// TIA Portal V17 export
// export: Created 2026-04-13T11:12:53.7703103Z, ExportSetting WithDefaults, DisplayName Totally Integrated Automation Portal, DisplayVersion V17 Update 4, DisplayName TIA Portal Openness, DisplayVersion V17 Update 4, DisplayName TIA Portal Version Control Interface, DisplayVersion V17, DisplayName SINAMICS Startdrive Advanced, DisplayVersion V17, DisplayName SINAMICS Startdrive G130, G150, S120, S150, SINAMICS MV, S210, DisplayVersion V17, DisplayName SINAMICS Startdrive G110M, G120, G120C, G120D, G120P, G115D, DisplayVersion V17, DisplayName STEP 7 Professional, DisplayVersion V17 Update 4, DisplayName STEP 7 Safety, DisplayVersion V17, DisplayName WinCC Professional, DisplayVersion V17 Update 4
TagTable "PV"
  PV_JF进风温度 : Real  (PLC tag PV.JF进风温度, HMI_连接_1, 1 s)
  PV_JF进风温度写读 : Real  (PLC tag PV.JF进风温度写读, HMI_连接_1, 1 s)
  PV_CF出风温度 : Real  (PLC tag PV.CF出风温度, HMI_连接_1, 1 s)
  PV_WQ尾气温度 : Real  (PLC tag PV.WQ尾气温度, HMI_连接_1, 1 s)
  PV_JF进风温度P : Real  (PLC tag PV.JF进风温度P, HMI_连接_1, 1 s)
  PV_JF进风温度I : Real  (PLC tag PV.JF进风温度I, HMI_连接_1, 1 s)
  PV_JF进风温度D : Real  (PLC tag PV.JF进风温度D, HMI_连接_1, 1 s)
  PV_SF送风机 : Real  (PLC tag PV.SF送风机, HMI_连接_1, 1 s)
  PV_YF引风机 : Real  (PLC tag PV.YF引风机, HMI_连接_1, 1 s)
  PV_LX离心雾化器 : Real  (PLC tag PV.LX离心雾化器, HMI_连接_1, 1 s)
  PV_LX离心雾化油压 : Real  (PLC tag PV.LX离心雾化油压, HMI_连接_1, 1 s)
  PV_JL进料泵 : Real  (PLC tag PV.JL进料泵, HMI_连接_1, 1 s)
  PV_JL进料压力 : Real  (PLC tag PV.JL进料压力, HMI_连接_1, 1 s)
  PV_JL进料流量 : Real  (PLC tag PV.JL进料流量, HMI_连接_1, 1 s)
  PV_JF进风流量计 : Real  (PLC tag PV.JF进风流量计, HMI_连接_1, 1 s)
  PV_YH氧含仪1 : Real  (PLC tag PV.YH氧含仪1, HMI_连接_1, 1 s)
  PV_YH氧含仪2 : Real  (PLC tag PV.YH氧含仪2, HMI_连接_1, 1 s)
  PV_JF进风压差变送器 : Real  (PLC tag PV.JF进风压差变送器, HMI_连接_1, 1 s)
  PV_BD布袋压差变送器 : Real  (PLC tag PV.BD布袋压差变送器, HMI_连接_1, 1 s)
  PV_CF出风高效压差变送器 : Real  (PLC tag PV.CF出风高效压差变送器, HMI_连接_1, 1 s)
  PV_SF输送高效压差变送器 : Real  (PLC tag PV.SF输送高效压差变送器, HMI_连接_1, 1 s)
  PV_TN塔内压力 : Real  (PLC tag PV.TN塔内压力, HMI_连接_1, 1 s)
  PV_GD管道压力变送器 : Real  (PLC tag PV.GD管道压力变送器, HMI_连接_1, 1 s)
  PV_JD进氮压力 : Real  (PLC tag PV.JD进氮压力, HMI_连接_1, 1 s)
  PV_YJ一级溶剂液位计 : Real  (PLC tag PV.YJ一级溶剂液位计, HMI_连接_1, 1 s)
  PV_EJ二级溶剂液位计 : Real  (PLC tag PV.EJ二级溶剂液位计, HMI_连接_1, 1 s)
  PV_CW除雾溶剂液位计 : Real  (PLC tag PV.CW除雾溶剂液位计, HMI_连接_1, 1 s)
  PV_HF回风加热比例反馈 : Real  (PLC tag PV.HF回风加热比例反馈, HMI_连接_1, 1 s)
  PV_JF进风加热比例反馈 : Real  (PLC tag PV.JF进风加热比例反馈, HMI_连接_1, 1 s)
  PV_FK放空比例反馈 : Real  (PLC tag PV.FK放空比例反馈, HMI_连接_1, 1 s)
  PV_HF回风温度 : Real  (PLC tag PV.HF回风温度, HMI_连接_1, 1 s)
  PV_SS输送温度 : Real  (PLC tag PV.SS输送温度, HMI_连接_1, 1 s)
  PV_FD阀导气压 : Real  (PLC tag PV.FD阀导气压, HMI_连接_1, 1 s)
  PV_SS输送温度P : Real  (PLC tag PV.SS输送温度P, HMI_连接_1, 1 s)
  PV_SS输送温度I : Real  (PLC tag PV.SS输送温度I, HMI_连接_1, 1 s)
  PV_SS输送温度D : Real  (PLC tag PV.SS输送温度D, HMI_连接_1, 1 s)
  PV_HF回风温度P : Real  (PLC tag PV.HF回风温度P, HMI_连接_1, 1 s)
  PV_HF回风温度I : Real  (PLC tag PV.HF回风温度I, HMI_连接_1, 1 s)
  PV_HF回风温度D : Real  (PLC tag PV.HF回风温度D, HMI_连接_1, 1 s)
  PV_JL进料平均流量 : Real  (PLC tag PV.JL进料平均流量, HMI_连接_1, 1 s)
  PV_JS碱水出压 : Real  (PLC tag PV.JS碱水出压, HMI_连接_1, 1 s)
  PV_JS碱水温度 : Real  (PLC tag PV.JS碱水温度, HMI_连接_1, 1 s)
  PV_RJ溶剂出压 : Real  (PLC tag PV.RJ溶剂出压, HMI_连接_1, 1 s)
  PV_HF回风加热开度 : Real  (PLC tag PV.HF回风加热开度, HMI_连接_1, 1 s)
  PV_SC四参数当前模式 : Int  (PLC tag PV.SC四参数当前模式, HMI_连接_1, 1 s)
  PV_JL进料当前模式 : Int  (PLC tag PV.JL进料当前模式, HMI_连接_1, 1 s)
  PV_DJ电加热开度 : Real  (PLC tag PV.DJ电加热开度, HMI_连接_1, 1 s)
  PV_SS输送加热开度 : Real  (PLC tag PV.SS输送加热开度, HMI_连接_1, 1 s)
  PV_QZ前置液位 : Real  (PLC tag PV.QZ前置液位, HMI_连接_1, 1 s)
  PV_TJ调节时间显示 : Real  (PLC tag PV.TJ调节时间显示, HMI_连接_1, 1 s)
  PV_JS碱水液位 : Real  (PLC tag PV.JS碱水液位, HMI_连接_1, 1 s)
  PV_CS纯水温度 : Real  (PLC tag PV.CS纯水温度, HMI_连接_1, 1 s)
  PV_CS纯水液位 : Real  (PLC tag PV.CS纯水液位, HMI_连接_1, 1 s)
  PV_RJ溶剂温度 : Real  (PLC tag PV.RJ溶剂温度, HMI_连接_1, 1 s)
  PV_RJ溶剂液位 : Real  (PLC tag PV.RJ溶剂液位, HMI_连接_1, 1 s)
  PV_JC碱纯压力 : Real  (PLC tag PV.JC碱纯压力, HMI_连接_1, 1 s)
  PV_CS纯水压力 : Real  (PLC tag PV.CS纯水压力, HMI_连接_1, 1 s)
